// Mitsubishi GX Works2 project: 램프3   PLC: Q02/Q02H

PROGRAM MAIN
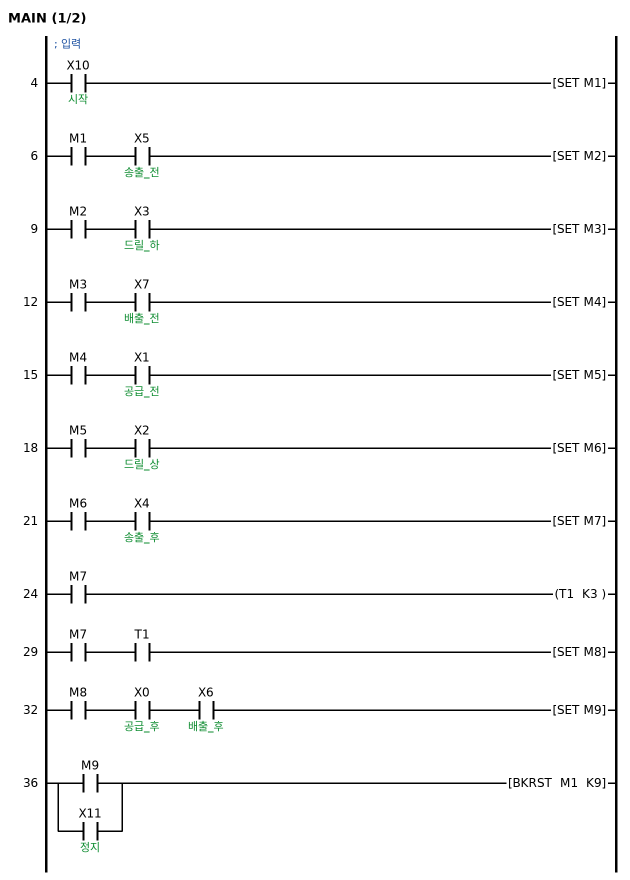
; 입력
4     LD      X10  ; 시작
      SET     M1
6     LD      M1
      AND     X5  ; 송출_전
      SET     M2
9     LD      M2
      AND     X3  ; 드릴_하
      SET     M3
12    LD      M3
      AND     X7  ; 배출_전
      SET     M4
15    LD      M4
      AND     X1  ; 공급_전
      SET     M5
18    LD      M5
      AND     X2  ; 드릴_상
      SET     M6
21    LD      M6
      AND     X4  ; 송출_후
      SET     M7
24    LD      M7
      OUT     T1 K3
29    LD      M7
      AND     T1
      SET     M8
32    LD      M8
      AND     X0  ; 공급_후
      AND     X6  ; 배출_후
      SET     M9
36    LD      M9
      OR      X11  ; 정지
      BKRST   M1 K9
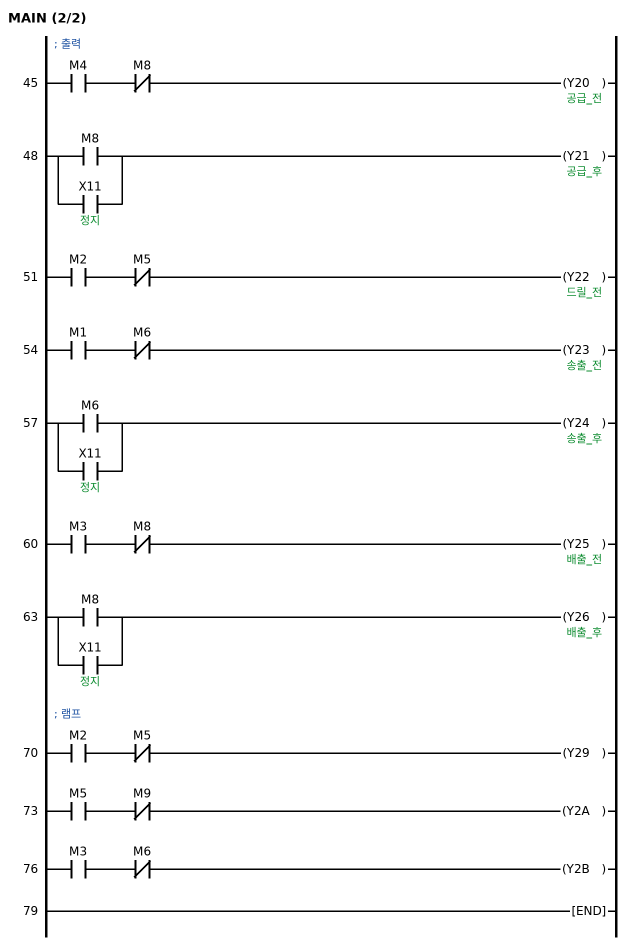
; 출력
45    LD      M4
      ANI     M8
      OUT     Y20  ; 공급_전
48    LD      M8
      OR      X11  ; 정지
      OUT     Y21  ; 공급_후
51    LD      M2
      ANI     M5
      OUT     Y22  ; 드릴_전
54    LD      M1
      ANI     M6
      OUT     Y23  ; 송출_전
57    LD      M6
      OR      X11  ; 정지
      OUT     Y24  ; 송출_후
60    LD      M3
      ANI     M8
      OUT     Y25  ; 배출_전
63    LD      M8
      OR      X11  ; 정지
      OUT     Y26  ; 배출_후
; 램프
70    LD      M2
      ANI     M5
      OUT     Y29
73    LD      M5
      ANI     M9
      OUT     Y2A
76    LD      M3
      ANI     M6
      OUT     Y2B
79    END
END_PROGRAM
